Universal Robots PolyScope program: ur5_control.urp

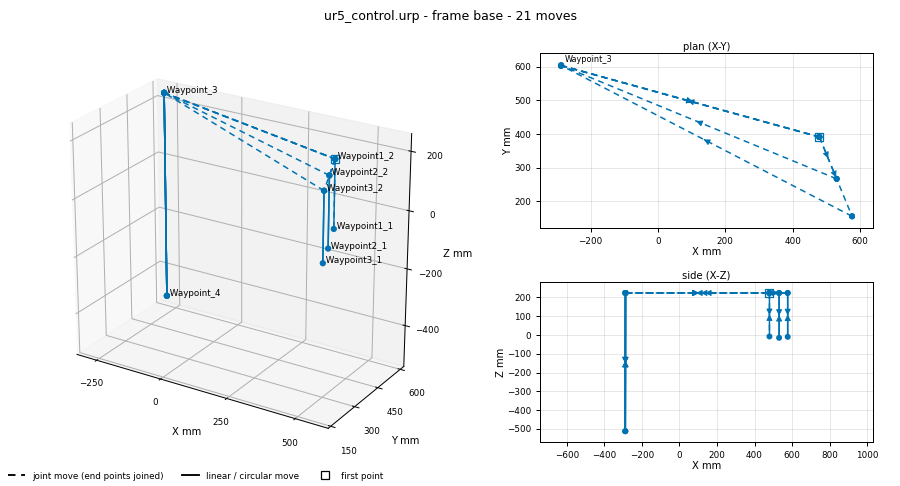
[picture p0: tool path of ur5_control.urp in frame base, 21 of 21 moves have a stored position in this frame; points joined in program order, loops and branches not executed]
Program ur5_control (installation=default directory=/ursim/programs createdIn=5.21.3 lastSavedIn=5.21.3 robotSerialNumber=20195599999)
Calibrated DH parameters: a=[0, -0.425, -0.3922, 0, 0, 0]; d=[0.1625, 0, 0, 0.1333, 0.0997, 0.0996]; alpha=[1.570796, 0, 0, 1.570796, -1.570796, 0]; deltaTheta=[0, 0, 0, 0, 0, 0]
InitVariablesNode
Robot Program (runOnlyOnce=false)
  MoveJ speed 60 deg/s, acceleration 80 deg/s^2 (useActiveTCP=true optimoveEnabled=false optiMoveSpeed=0.3 optiMoveAcceleration=0.09) feature=Base
    Waypoint Waypoint1_2: TCP in base x=479.522 y=391.169 z=224.12 mm, rx=-2.5592 ry=1.7142 rz=0.0947 rad; joints [-154.02, -64.91, 100.12, 233.59, -85.23, 3.66] deg
  Wait Sleep waitTime=3
  MoveJ speed 60 deg/s, acceleration 80 deg/s^2 (useActiveTCP=true optimoveEnabled=false optiMoveSpeed=0.3 optiMoveAcceleration=0.09) feature=Base
    Waypoint Waypoint1_1: TCP in base x=479.65 y=391.039 z=-7.708 mm, rx=-2.5601 ry=1.7145 rz=0.0924 rad; joints [-154.02, -40.58, 103.6, 205.78, -85.33, 3.65] deg
  Wait Sleep waitTime=0.5
  MoveL speed 250 mm/s, acceleration 1200 mm/s^2 (useActiveTCP=true optimoveEnabled=false optiMoveSpeed=0.3 optiMoveAcceleration=0.09) feature=Base
    Waypoint Waypoint1_2: TCP in base x=479.522 y=391.169 z=224.12 mm, rx=-2.5592 ry=1.7142 rz=0.0947 rad; joints [-154.02, -64.91, 100.12, 233.59, -85.23, 3.66] deg
  Wait Sleep waitTime=0.5
  MoveJ speed 60 deg/s, acceleration 80 deg/s^2 (useActiveTCP=true optimoveEnabled=false optiMoveSpeed=0.3 optiMoveAcceleration=0.09) feature=Base
    Waypoint Waypoint_3: TCP in base x=-287.168 y=603.408 z=224.159 mm, rx=-2.5354 ry=1.7009 rz=-0.0647 rad; joints [-75.24, -58.79, 90.36, 236.92, -95.38, 82.4] deg
  Wait Sleep waitTime=0.5
  MoveL speed 250 mm/s, acceleration 1200 mm/s^2 (useActiveTCP=true optimoveEnabled=false optiMoveSpeed=0.3 optiMoveAcceleration=0.09) feature=Base
    Waypoint Waypoint_4: TCP in base x=-288.037 y=603.108 z=-512.12 mm, rx=-2.5364 ry=1.6993 rz=-0.0646 rad; joints [-75.16, 35.24, 22.84, 210.41, -95.38, 82.41] deg; TCP offset x=0 y=0 z=0 mm, rx=0 ry=0 rz=0 rad
  Wait Sleep waitTime=0.5
  MoveL speed 250 mm/s, acceleration 1200 mm/s^2 (useActiveTCP=true optimoveEnabled=false optiMoveSpeed=0.3 optiMoveAcceleration=0.09) feature=Base
    Waypoint Waypoint_3: TCP in base x=-287.168 y=603.408 z=224.159 mm, rx=-2.5354 ry=1.7009 rz=-0.0647 rad; joints [-75.24, -58.79, 90.36, 236.92, -95.38, 82.4] deg
  Wait Sleep waitTime=0.5
  MoveJ speed 60 deg/s, acceleration 80 deg/s^2 (useActiveTCP=true optimoveEnabled=false optiMoveSpeed=0.3 optiMoveAcceleration=0.09) feature=Base
    Waypoint Waypoint1_2: TCP in base x=479.522 y=391.169 z=224.12 mm, rx=-2.5592 ry=1.7142 rz=0.0947 rad; joints [-154.02, -64.91, 100.12, 233.59, -85.23, 3.66] deg
  Wait Sleep waitTime=3
  MoveJ speed 60 deg/s, acceleration 80 deg/s^2 (useActiveTCP=true optimoveEnabled=false optiMoveSpeed=0.3 optiMoveAcceleration=0.09) feature=Base
    Waypoint Waypoint2_2: TCP in base x=530.932 y=266.908 z=224.126 mm, rx=-2.5588 ry=1.7141 rz=0.0943 rad; joints [-167.12, -67.69, 104.05, 233.53, -85.08, -9.48] deg
  Wait Sleep waitTime=0.5
  MoveL speed 250 mm/s, acceleration 1200 mm/s^2 (useActiveTCP=true optimoveEnabled=false optiMoveSpeed=0.3 optiMoveAcceleration=0.09) feature=Base
    Waypoint Waypoint2_1: TCP in base x=531.03 y=266.735 z=-14.737 mm, rx=-2.5601 ry=1.7147 rz=0.0921 rad; joints [-167.12, -41.34, 107.56, 203.67, -85.19, -9.49] deg
  Wait Sleep waitTime=0.5
  MoveL speed 250 mm/s, acceleration 1200 mm/s^2 (useActiveTCP=true optimoveEnabled=false optiMoveSpeed=0.3 optiMoveAcceleration=0.09) feature=Base
    Waypoint Waypoint2_2: TCP in base x=530.932 y=266.908 z=224.126 mm, rx=-2.5588 ry=1.7141 rz=0.0943 rad; joints [-167.12, -67.69, 104.05, 233.53, -85.08, -9.48] deg
  Wait Sleep waitTime=0.5
  MoveJ speed 60 deg/s, acceleration 80 deg/s^2 (useActiveTCP=true optimoveEnabled=false optiMoveSpeed=0.3 optiMoveAcceleration=0.09) feature=Base
    Waypoint Waypoint_3: TCP in base x=-287.168 y=603.408 z=224.159 mm, rx=-2.5354 ry=1.7009 rz=-0.0647 rad; joints [-75.24, -58.79, 90.36, 236.92, -95.38, 82.4] deg
  Wait Sleep waitTime=0.5
  MoveL speed 250 mm/s, acceleration 1200 mm/s^2 (useActiveTCP=true optimoveEnabled=false optiMoveSpeed=0.3 optiMoveAcceleration=0.09) feature=Base
    Waypoint Waypoint_4: TCP in base x=-288.037 y=603.108 z=-512.12 mm, rx=-2.5364 ry=1.6993 rz=-0.0646 rad; joints [-75.16, 35.24, 22.84, 210.41, -95.38, 82.41] deg; TCP offset x=0 y=0 z=0 mm, rx=0 ry=0 rz=0 rad
  Wait Sleep waitTime=0.5
  MoveL speed 250 mm/s, acceleration 1200 mm/s^2 (useActiveTCP=true optimoveEnabled=false optiMoveSpeed=0.3 optiMoveAcceleration=0.09) feature=Base
    Waypoint Waypoint_3: TCP in base x=-287.168 y=603.408 z=224.159 mm, rx=-2.5354 ry=1.7009 rz=-0.0647 rad; joints [-75.24, -58.79, 90.36, 236.92, -95.38, 82.4] deg
  Wait Sleep waitTime=0.5
  MoveJ speed 60 deg/s, acceleration 80 deg/s^2 (useActiveTCP=true optimoveEnabled=false optiMoveSpeed=0.3 optiMoveAcceleration=0.09) feature=Base
    Waypoint Waypoint1_2: TCP in base x=479.522 y=391.169 z=224.12 mm, rx=-2.5592 ry=1.7142 rz=0.0947 rad; joints [-154.02, -64.91, 100.12, 233.59, -85.23, 3.66] deg
  Wait Sleep waitTime=3
  MoveJ speed 60 deg/s, acceleration 80 deg/s^2 (useActiveTCP=true optimoveEnabled=false optiMoveSpeed=0.3 optiMoveAcceleration=0.09) feature=Base
    Waypoint Waypoint3_2: TCP in base x=576.697 y=155.655 z=224.032 mm, rx=-2.5589 ry=1.7139 rz=0.0945 rad; joints [-178.62, -67.27, 103.12, 235.03, -85.15, -21.03] deg; TCP offset x=0 y=0 z=0 mm, rx=0 ry=0 rz=0 rad
  Wait Sleep waitTime=0.5
  MoveL speed 250 mm/s, acceleration 1200 mm/s^2 (useActiveTCP=true optimoveEnabled=false optiMoveSpeed=0.3 optiMoveAcceleration=0.09) feature=Base
    Waypoint Waypoint3_1: TCP in base x=576.77 y=155.466 z=-9.623 mm, rx=-2.5602 ry=1.7148 rz=0.0928 rad; joints [-178.62, -41.93, 106.89, 205.92, -85.26, -21.03] deg
  Wait Sleep waitTime=0.5
  MoveL speed 250 mm/s, acceleration 1200 mm/s^2 (useActiveTCP=true optimoveEnabled=false optiMoveSpeed=0.3 optiMoveAcceleration=0.09) feature=Base
    Waypoint Waypoint3_2: TCP in base x=576.697 y=155.655 z=224.032 mm, rx=-2.5589 ry=1.7139 rz=0.0945 rad; joints [-178.62, -67.27, 103.12, 235.03, -85.15, -21.03] deg; TCP offset x=0 y=0 z=0 mm, rx=0 ry=0 rz=0 rad
  Wait Sleep waitTime=0.5
  MoveJ speed 60 deg/s, acceleration 80 deg/s^2 (useActiveTCP=true optimoveEnabled=false optiMoveSpeed=0.3 optiMoveAcceleration=0.09) feature=Base
    Waypoint Waypoint_3: TCP in base x=-287.168 y=603.408 z=224.159 mm, rx=-2.5354 ry=1.7009 rz=-0.0647 rad; joints [-75.24, -58.79, 90.36, 236.92, -95.38, 82.4] deg
  Wait Sleep waitTime=0.5
  MoveL speed 250 mm/s, acceleration 1200 mm/s^2 (useActiveTCP=true optimoveEnabled=false optiMoveSpeed=0.3 optiMoveAcceleration=0.09) feature=Base
    Waypoint Waypoint_4: TCP in base x=-288.037 y=603.108 z=-512.12 mm, rx=-2.5364 ry=1.6993 rz=-0.0646 rad; joints [-75.16, 35.24, 22.84, 210.41, -95.38, 82.41] deg; TCP offset x=0 y=0 z=0 mm, rx=0 ry=0 rz=0 rad
  Wait Sleep waitTime=0.5
  MoveL speed 250 mm/s, acceleration 1200 mm/s^2 (useActiveTCP=true optimoveEnabled=false optiMoveSpeed=0.3 optiMoveAcceleration=0.09) feature=Base
    Waypoint Waypoint_3: TCP in base x=-287.168 y=603.408 z=224.159 mm, rx=-2.5354 ry=1.7009 rz=-0.0647 rad; joints [-75.24, -58.79, 90.36, 236.92, -95.38, 82.4] deg
  Wait Sleep waitTime=0.5
  MoveJ speed 60 deg/s, acceleration 80 deg/s^2 (useActiveTCP=true optimoveEnabled=false optiMoveSpeed=0.3 optiMoveAcceleration=0.09) feature=Base
    Waypoint Waypoint1_2: TCP in base x=479.522 y=391.169 z=224.12 mm, rx=-2.5592 ry=1.7142 rz=0.0947 rad; joints [-154.02, -64.91, 100.12, 233.59, -85.23, 3.66] deg
  Wait Sleep waitTime=3
